# EPICS substitutions: iocs/MC02/db/SAI_8MotorStatus.substitutions
file /opt/epics/modules/SAI/db/SAI_8MotorStatus.db {
    pattern {	ASYNPORT,	TMOT,		SCAN,		P,		R}
        { 	"pmac",		"1",		".2 second",	"XF:06BMA-OP","{MC:02}"}
}

#Sample naming - XF:06BMA-OP{Mono:DCM1-Ax:Bragg}Mtr
